SUBAPPLICATION Aux_IE_1 (* 1 AuxFunction2-Objekt, liest ein konfigurierbares Event (AuxiliaryState, z.B. AuxEnabled) als reines IND-Event - duenner Wrapper um Aux_IE, analog zu Softkey_IE_1 (Konvention in diesem Projekt: die isobus-IE-Bausteine werden nie roh inline verwendet, immer gewrappt). *)
  (* Standard: 61499-2 *)
  (* Version 1.0, 2026-09-11, Franz Höpfinger, initial implementation *)
  PACKAGE MyLib::sys;
  IMPORT isobus::UT::Q::const::IDs::ID_NULL;
  IMPORT isobus::UT::io::Auxiliary::IN::AuxiliaryState::Invalid;
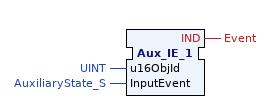
  EVENT_OUTPUT
    IND; (* Feuert wenn das konfigurierte InputEvent auftritt *)
  END_EVENT
  VAR_INPUT
    u16ObjId : UINT := ID_NULL; (* Object ID AuxFunction2 *)
    InputEvent : isobus::UT::io::Auxiliary::IN::AuxiliaryState_S := Invalid; (* z.B. AuxEnabled, AuxDisabled *)
  END_VAR
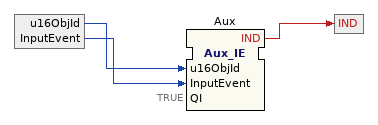
  FBS
    Aux : isobus::UT::io::Auxiliary::IN::Aux_IE(QI := TRUE);
  END_FBS
  EVENT_CONNECTIONS
    Aux.IND TO IND;
  END_CONNECTIONS
  DATA_CONNECTIONS
    u16ObjId TO Aux.u16ObjId;
    InputEvent TO Aux.InputEvent;
  END_CONNECTIONS
END_SUBAPPLICATION
